INTERFACE I_PosStation

METHOD EnableRequest : BOOL
VAR_INPUT
	OnOff : BOOL;
END_VAR
END_METHOD

PROPERTY InPosition : BOOL
GET
END_GET
END_PROPERTY

PROPERTY Linked : BOOL
GET
END_GET
END_PROPERTY

METHOD MoverChangeStep : BOOL
VAR_INPUT
	step : UDINT;
END_VAR
END_METHOD

PROPERTY RequestedStep : INT
SET
END_SET
END_PROPERTY

METHOD SetAttractStep : BOOL
VAR_INPUT
	step : INT;
END_VAR
END_METHOD

END_INTERFACE

(* stored: Version 1.1.0.1
   Itf I_PosStation: Id {bb604d4c-e6cd-4128-9a70-0d2422fff6af}
   Method EnableRequest: Id {058d8b3b-7bb9-49c0-b13c-b097a4571105}
   Property InPosition: Id {bf8a15f9-bff6-4784-b683-69069cd88e69}
   Get Get: Id {afb139da-a1bb-4421-8ea2-fe5dee3f7b56}
   Property Linked: Id {04d8bf98-113e-468c-b48e-f96b51b75d50}
   Get Get: Id {253d21f6-64d0-41cf-a2f1-5d121ea2a9a6}
   Method MoverChangeStep: Id {c47ed53a-e3e7-472b-86ef-d81b8a5b13ce}
   Property RequestedStep: Id {cc77b5be-5c81-4526-9224-f8271f42e456}
   Set Set: Id {9b67bfe0-375e-4621-aad7-3251c845e514}
   Method SetAttractStep: Id {e2b7f86c-fcda-489e-b91b-be6518d81640} *)
